(* IEC 61131-3 sources: CODESYS-IO-Visualization/CODESYS-IO-Visualization.fbsproj/Subs/Equipment, 8 files *)

(* ---- GetModbusCommStateString.fn.st ---- *)
FUNCTION GetModbusCommStateString : WSTRING(256)

VAR_INPUT
	State: INT;
END_VAR

VAR
	StateString: WSTRING(256);
END_VAR

CASE State OF
	0: StateString := "OFF";
	1: StateString := "Connecting";
	2: StateString := "Connected";
	3: StateString := "Disconnecting";
	4: StateString := "Socket Error";
ELSE
	StateString := "Unknown";
END_CASE;

GetModbusCommStateString := StateString;

(* ---- GetModbusDeviceStatusString.fn.st ---- *)
FUNCTION GetModbusDeviceStatusString : WSTRING(256)

VAR_INPUT
	ErrorCode: INT;
END_VAR

VAR
	ErrorString: WSTRING(256);
END_VAR

CASE ErrorCode OF
	0: ErrorString := "OK";
	1: ErrorString := "Illegal Function";
	2: ErrorString := "Illegal Data Address";
	3: ErrorString := "Illegal Data Value";
	4: ErrorString := "Slave Device Failure";
	5: ErrorString := "Acknowledge";
	6: ErrorString := "Slave Device Busy";
	7: ErrorString := "Memory Parity Error";
	8: ErrorString := "Gateway Path Unavailable";
	9: ErrorString := "Gateway Device Failed To Respond";
	10: ErrorString := "Response Timeout";
	11: ErrorString := "Response CRC Fail";
	12: ErrorString := "Response Wrong Slave";
	13: ErrorString := "Response Wrong Function Code";
	14: ErrorString := "TCP Communication Error";
	15: ErrorString := "Response Invalid Data";
	16: ErrorString := "Response Invalid Protocol";
	17: ErrorString := "Response Invalid Header";
	18: ErrorString := "Undefined";
ELSE
	ErrorString := "Error: Unknown";
END_CASE;

GetModbusDeviceStatusString := ErrorString;

(* ---- Equip.prg.st ---- *)
PROGRAM Equip

VAR_IN_OUT
	Data: Equip_UDT;
END_VAR

VAR
	i: INT;
END_VAR

// Enable Persist Storage
IF (Data.PersistSize = 0) THEN
	Data.PersistSize := SIZEOF(Equip_UDT);
END_IF;

// Clear Common Alarm Flags
Data.NotReadyActive := FALSE;
Data.InterlockActive := FALSE;
Data.FailureActive := FALSE;
Data.WarningActive := FALSE;
Data.TimerActive := FALSE;

//Alarms
AlarmDigital(alarm := Data.OOS);

Data.MaxSeverity := 0;
Data.AlarmLevel := 0;

FOR i := 0 TO 9 DO
	Data.Failure[i].Reset := Data.HMI.Reset;
	Data.Failure[i].OOS := Data.OOS.Active;
	AlarmDigital(alarm := Data.Failure[i]);
	IF (Data.Failure[i].Active) THEN
		Data.FailureActive := TRUE;
	END_IF;

	IF (Data.Failure[i].Severity > Data.MaxSeverity) THEN
		Data.MaxSeverity := Data.Failure[i].Severity;
	END_IF;

	IF (Data.Failure[i].AlarmLevel > 0) THEN
		IF (Data.AlarmLevel = 0) OR (Data.Failure[i].AlarmLevel < Data.AlarmLevel) THEN
			Data.AlarmLevel := Data.Failure[i].AlarmLevel;
		END_IF;
	END_IF;

	Data.Interlock[i].Reset := Data.HMI.Reset;
	Data.Interlock[i].OOS := Data.OOS.Active;
	AlarmDigital(alarm := Data.Interlock[i]);
	IF (Data.Interlock[i].Active) THEN
		Data.InterlockActive := TRUE;
	END_IF;

	IF (Data.Interlock[i].Severity > Data.MaxSeverity) THEN
		Data.MaxSeverity := Data.Interlock[i].Severity;
	END_IF;

	IF (Data.Interlock[i].AlarmLevel > 0) THEN
		IF (Data.AlarmLevel = 0) OR (Data.Interlock[i].AlarmLevel < Data.AlarmLevel) THEN
			Data.AlarmLevel := Data.Interlock[i].AlarmLevel;
		END_IF;
	END_IF;

	Data.NotReady[i].Reset := Data.HMI.Reset;
	Data.NotReady[i].OOS := Data.OOS.Active;
	AlarmDigital(alarm := Data.NotReady[i]);
	IF (Data.NotReady[i].Active) THEN
		Data.NotReadyActive := TRUE;
	END_IF;

	IF (Data.NotReady[i].Severity > Data.MaxSeverity) THEN
		Data.MaxSeverity := Data.NotReady[i].Severity;
	END_IF;

	IF (Data.NotReady[i].AlarmLevel > 0) THEN
		IF (Data.AlarmLevel = 0) OR (Data.NotReady[i].AlarmLevel < Data.AlarmLevel) THEN
			Data.AlarmLevel := Data.NotReady[i].AlarmLevel;
		END_IF;
	END_IF;

	Data.Warning[i].Reset := Data.HMI.Reset;
	Data.Warning[i].OOS := Data.OOS.Active;
	AlarmDigital(alarm := Data.Warning[i]);
	IF (Data.Warning[i].Active) THEN
		Data.WarningActive := TRUE;
	END_IF;

	IF (Data.Warning[i].Severity > Data.MaxSeverity) THEN
		Data.MaxSeverity := Data.Warning[i].Severity;
	END_IF;

	IF (Data.Warning[i].AlarmLevel > 0) THEN
		IF (Data.AlarmLevel = 0) OR (Data.Warning[i].AlarmLevel < Data.AlarmLevel) THEN
			Data.AlarmLevel := Data.Warning[i].AlarmLevel;
		END_IF;
	END_IF;

	IF (Data.Timer0[i].On) THEN
		Data.TimerActive := TRUE;
	END_IF;
END_FOR;

Data.ResetTimer.In := Data.HMI.Reset OR Data.PLC.Reset;
Timer(TimerData := Data.ResetTimer);

IF (Data.ResetTimer.Q) THEN
	Data.HMI.Reset := FALSE;
	Data.PLC.Reset := FALSE;
END_IF;

//Set Equipment Stats
Data.Stats.StatInput := Data.Running OR Data.Opened OR (NOT Data.Closed);
Data.Stats.OOSInput := Data.OOS.Active;
Data.Stats.AvailalbeInput := (NOT Data.NotReadyActive) AND (NOT Data.FailureActive) AND (NOT Data.InterlockActive) AND (NOT Data.OOS.Active);

Equip_Statistics(Data := Data.Stats);

(* ---- Equip_Statistics.prg.st ---- *)
PROGRAM Equip_Statistics

VAR_IN_OUT
	Data: Equip_Statistics_UDT;
END_VAR

// Process Runtime
Data.RuntimeCumulative.Enable := Data.StatInput;
Runtime(Data := Data.RuntimeCumulative);

Data.RuntimeDaily.Enable := Data.StatInput;
Runtime(Data := Data.RuntimeDaily);

Data.RuntimeMonthly.Enable := Data.StatInput;
Runtime(Data := Data.RuntimeMonthly);

// Process Available Time
Data.AvailableTime.Enable := Data.AvailalbeInput;
Runtime(Data := Data.AvailableTime);

Data.AvailableTimeDaily.Enable := Data.AvailalbeInput;
Runtime(Data := Data.AvailableTimeDaily);

Data.AvailableTimeMonthly.Enable := Data.AvailalbeInput;
Runtime(Data := Data.AvailableTimeMonthly);

// Process Out of Service Time
Data.OOSTime.Enable := Data.OOSInput;
Runtime(Data := Data.OOSTime);

Data.OOSTimeDaily.Enable := Data.OOSInput;
Runtime(Data := Data.OOSTimeDaily);

Data.OOSTimeMonthly.Enable := Data.OOSInput;
Runtime(Data := Data.OOSTimeMonthly);

// Process Starts
IF ((NOT Data.LastStat) AND Data.StatInput) THEN
	Data.StartsCumulative := Data.StartsCumulative + 1;
	Data.StartsToday := Data.StartsToday + 1;
	Data.StartsMonth := Data.StartsMonth + 1;
	Data.ActualStartsThisHour := Data.ActualStartsThisHour + 1;
END_IF;
Data.LastStat := Data.StatInput;

// Daily Stats
IF (Data.RuntimeDaily.ResetAccumulator AND (NOT Data.DailyResetDone)) THEN
	Data.StartsYesterday := Data.StartsToday;
	Data.StartsToday := 0;
	Data.DailyResetDone := TRUE;
END_IF;

IF (NOT Data.RuntimeDaily.ResetAccumulator) THEN
	Data.DailyResetDone := FALSE;
END_IF;

//Monthly Stats
IF (Data.RuntimeMonthly.ResetAccumulator AND (NOT Data.MonthlyResetDone)) THEN
	Data.StartsLastMonth := Data.StartsMonth;
	Data.StartsMonth := 0;
	Data.MonthlyResetDone := TRUE;
END_IF;

IF (NOT Data.RuntimeMonthly.ResetAccumulator) THEN
	Data.MonthlyResetDone := FALSE;
END_IF;

//Hour Stats
IF ((Lib_GVL.ClockLocal.Minute = 0) AND (Lib_GVL.ClockLocal.Second < 5)) THEN
	Data.ActualStartsThisHour := 0;
END_IF;

Data.ExcessiveStartsPerHour := (Data.ActualStartsThisHour > Data.StartsPerHourLimit);

(* ---- MapEquip_Simple.prg.st ---- *)
PROGRAM MapEquip_Simple

VAR_IN_OUT
	Equip: Equip_UDT;
END_VAR

VAR_INPUT
	Remote: BOOL;
	Running: BOOL;
	Failed: BOOL;
END_VAR

VAR_OUTPUT
	RunCmd: BOOL;
	FailureActive: BOOL;
END_VAR

// Map Inputs
Equip.Raw.BOOL0[0] := Remote;
Equip.Raw.BOOL0[1] := Running;
Equip.Raw.BOOL0[2] := Failed;

// Map Outputs
RunCmd := Equip.RunCmd OR Equip.OpenCmd;
FailureActive := Equip.FailureActive;

(* ---- MapEquip_Valve.prg.st ---- *)
PROGRAM MapEquip_Valve

VAR_IN_OUT
	Equip: Equip_UDT;
END_VAR

VAR_INPUT
	Remote: BOOL;
	GCPRemote: BOOL;
	Opened: BOOL;
	Closed: BOOL;
	Failed: BOOL;
	Alarm: BOOL;
	CommFail: BOOL;
	Position: REAL;
	OpenHS: BOOL;
	CloseHS: BOOL;
	Interlock1: BOOL;
	Interlock2: BOOL;
END_VAR

VAR_OUTPUT
	OpenCmd: BOOL;
	CloseCmd: BOOL;
END_VAR

// Map Inputs
MapEquip_Valve.Equip.Raw.BOOL0[0] := Remote;
MapEquip_Valve.Equip.Raw.BOOL0[6] := GCPRemote;
MapEquip_Valve.Equip.Raw.BOOL0[1] := Closed;
MapEquip_Valve.Equip.Raw.BOOL0[2] := Opened;
MapEquip_Valve.Equip.Raw.BOOL0[3] := Alarm;
MapEquip_Valve.Equip.Raw.BOOL0[4] := Failed;
MapEquip_Valve.Equip.Raw.BOOL0[7] := OpenHS;
MapEquip_Valve.Equip.Raw.BOOL0[8] := CloseHS;
MapEquip_Valve.Equip.Raw.REAL0[0] := Position;
MapEquip_Valve.Equip.Raw.BOOL0[5] := CommFail;
MapEquip_Valve.Equip.Raw.BOOL0[12] := Interlock1;
MapEquip_Valve.Equip.Raw.BOOL0[17] := Interlock2;

// Map Outputs
OpenCmd := MapEquip_Valve.Equip.OpenCmd;
CloseCmd := MapEquip_Valve.Equip.CloseCmd;

(* ---- MapValveEquipFromRotork.prg.st ---- *)
PROGRAM MapValveEquipFromRotork

VAR_IN_OUT
	Valve: Equip_UDT;
	MB: RotorkValve_UDT;
END_VAR

Valve.Raw.SWITCH0[0] := WORD_TO_INT(MB.InputReg00);
Valve.Raw.BOOL0[0] := MB.Actuator_Moving;
Valve.Raw.BOOL0[1] := MB.Valve_Closed;
Valve.Raw.BOOL0[2] := MB.Valve_Opened;
Valve.Raw.BOOL0[3] := MB.Running_Closed;
Valve.Raw.BOOL0[4] := MB.Running_Open;
Valve.Raw.BOOL0[5] := MB.Remote_Selected;
Valve.Raw.BOOL0[6] := MB.Local_Stop_Selected_Offline;
Valve.Raw.BOOL0[7] := MB.Local_Stop_Selected;
Valve.Raw.BOOL0[8] := MB.Thermostat_Tripped;
Valve.Raw.BOOL0[9] := MB.Monitor_Relay;
Valve.Raw.BOOL0[10] := MB.Valve_Obstructed;
Valve.Raw.BOOL0[11] := MB.Valve_Jammed;
Valve.Raw.BOOL0[12] := MB.Valve_Moving_By_Hand;
Valve.Raw.BOOL0[13] := MB.Moving_Inhibited_by_MIT;
Valve.Raw.BOOL0[14] := MB.Position_Control_Enabled;
Valve.Raw.BOOL0[15] := MB.EEPROM_Checksum_Failure;

Valve.Raw.SWITCH0[1] := WORD_TO_INT(MB.InputReg01);
Valve.Raw.BOOL0[20] := MB.Battery_Low;
Valve.Raw.BOOL0[21] := MB.Open_Interlock_Active;
Valve.Raw.BOOL0[22] := MB.Close_Interlock_Active;
Valve.Raw.BOOL0[23] := MB.DI_1;
Valve.Raw.BOOL0[24] := MB.DI_2;
Valve.Raw.BOOL0[25] := MB.DI_3;
Valve.Raw.BOOL0[26] := MB.DI_4;
Valve.Raw.BOOL0[27] := MB.Reserved_7;
Valve.Raw.BOOL0[28] := MB.Reserved_8;
Valve.Raw.BOOL0[29] := MB.Reserved_9;
Valve.Raw.BOOL0[30] := MB.Control_Contention;
Valve.Raw.BOOL0[31] := MB.Partial_Stroke_Test_in_Progress;
Valve.Raw.BOOL0[32] := MB.Partial_Stroke_Test_Error;
Valve.Raw.BOOL0[33] := MB.General_Alarm;
Valve.Raw.BOOL0[34] := MB.Reserved_14;
Valve.Raw.BOOL0[35] := MB.Reserved_15;

Valve.Raw.REAL0[0] := MB.Valve_Position;
Valve.Raw.REAL0[1] := MB.Actuator_Torque;
Valve.Raw.REAL0[2] := MB.Analog_Input;

MB.Actuator_Position_Command := Valve.PositionCmd;

MB.Actuator_Control := 0;
IF (Valve.OpenCmd) THEN
	MB.Actuator_Control := 2;
END_IF;
IF (Valve.CloseCmd) THEN
	MB.Actuator_Control := 1;
END_IF;

MB.SignalLossAction := Valve.Raw.SWITCH0[50];
MB.SignalLossPosition := Valve.Raw.SWITCH0[51];

Valve.Raw.REAL0[40] := DINT_TO_REAL(MB.Status);
Valve.Raw.SWITCH0[40] := UINT_TO_INT(MB.SlaveState);
Valve.Raw.SWITCH0[41] := MB.SlaveErrorCode;
Valve.Raw.BOOL0[40] := MB.SlaveError;
Valve.Raw.BOOL0[41] := MB.CI;
Valve.Raw.BOOL0[42] := (MB.SlaveState <> 2) OR MB.SlaveError OR (MB.SlaveErrorCode <> 0); // Slave Comm as failed
Valve.Raw.STRING0[0] := GetModbusDeviceStatusString(ErrorCode := MB.SlaveErrorCode);
Valve.Raw.STRING0[1] := GetModbusCommStateString(State := UINT_TO_INT(MB.SlaveState));

// Set Simulator Data from HMI Data in Equipment_Valve
MB.Simulator.Thermostat_Tripped := Valve.HMI.BOOL0[75];
MB.Simulator.Monitor_Relay := Valve.HMI.BOOL0[76];
MB.Simulator.Valve_Obstructed := Valve.HMI.BOOL0[77];
MB.Simulator.Valve_Jammed := Valve.HMI.BOOL0[78];
MB.Simulator.Valve_Moving_By_Hand := Valve.HMI.BOOL0[79];
MB.Simulator.Moving_Inhibited_by_MIT := Valve.HMI.BOOL0[80];
MB.Simulator.Postion_Control_Enabled := Valve.HMI.BOOL0[81];
MB.Simulator.EEPROM_Checksum_Failure := Valve.HMI.BOOL0[82];
MB.Simulator.Battery_Low := Valve.HMI.BOOL0[83];
MB.Simulator.Open_Interlock_Active := Valve.HMI.BOOL0[84];
MB.Simulator.Close_Interlock_Active := Valve.HMI.BOOL0[85];
MB.Simulator.DI_1 := Valve.HMI.BOOL0[86];
MB.Simulator.DI_2 := Valve.HMI.BOOL0[87];
MB.Simulator.DI_3 := Valve.HMI.BOOL0[88];
MB.Simulator.DI_4 := Valve.HMI.BOOL0[89];
MB.Simulator.Reserved_7 := Valve.HMI.BOOL0[90];
MB.Simulator.Reserved_8 := Valve.HMI.BOOL0[91];
MB.Simulator.Reserved_9 := Valve.HMI.BOOL0[92];
MB.Simulator.Control_Contention := Valve.HMI.BOOL0[93];
MB.Simulator.Partial_Stroke_Test_in_Progress := Valve.HMI.BOOL0[94];
MB.Simulator.Partial_Stroke_Test_Error := Valve.HMI.BOOL0[95];
MB.Simulator.General_Alarm := Valve.HMI.BOOL0[96];
MB.Simulator.Reserved_14 := Valve.HMI.BOOL0[97];
MB.Simulator.Reserved_15 := Valve.HMI.BOOL0[98];
MB.Simulator.ibAuto := Valve.HMI.BOOL0[99];
MB.SimulationEnable := NOT Valve.HMI.BOOL0[100];

MB.Simulator.Analog_Input := Valve.HMI.REAL0[21];

MB.Simulator.InputData.Error := Valve.HMI.BOOL0[40];
MB.Simulator.InputData.State := INT_TO_UINT(Valve.HMI.SWITCH0[40]);
MB.Simulator.InputData.ErrorCode := DINT_TO_INT(Valve.HMI.SWITCH0[41]);

(* ---- Runtime.prg.st ---- *)
PROGRAM Runtime

VAR_IN_OUT
	Data: Runtime_UDT;
END_VAR

Data.ValueIn_Realtime := 1.0;
Data.Gain := 1.0;
Data.Timebase := 3600.0;
Data.Mode := 0;

Accum(Data := Data);
